(* IEC 61131-3 sources: CodesysTest/export/Testing/Actuators/FB_PneumaticVerticalActuator.pou, 1 file *)

(* ---- FB_PneumaticVerticalActuator.pou.st ---- *)
(*#-#-#-#-#-#-#-#-#-#---Declaration---#-#-#-#-#-#-#-#-#-#-#-#-#*)

FUNCTION_BLOCK FB_PneumaticVerticalActuator EXTENDS FB_PneumaticActuator IMPLEMENTS IUpDown
VAR_INPUT
	cylinder : ICylinder;
END_VAR
VAR_OUTPUT
END_VAR
VAR
END_VAR
VAR_IN_OUT
END_VAR
(*#-#-#-#-#-#-#-#-#-#---Implementation---#-#-#-#-#-#-#-#-#-#-#-#-#*)

//	Function Block: FB_PneumaticVerticalActuator
//	Description: Wrapper for a cylinder with Up/Down substitiuted for Extend/Retract
//
//
//	Usage:
//
//	Created by: Ben Hess
//	Created Date: 6-27-2019

EnableSimulation(cylinder, _simulateActive);
